SUBAPPLICATION Uebung_060 (* DigitalInput_I1 auf DigitalOutput_Q1 *)
  (* Standard: 61499-2 *)
  (* Version 1.0, 2023-10-23, franz *)
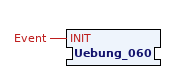
  EVENT_INPUT
    INIT;
  END_EVENT
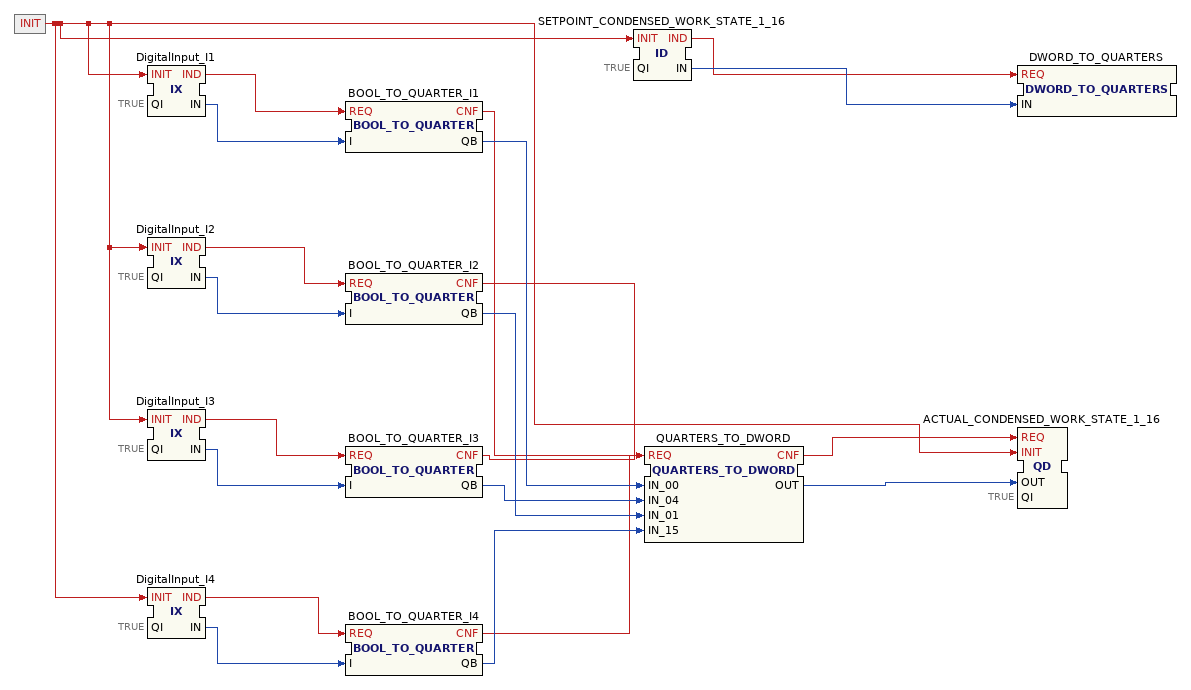
  FBS
    SETPOINT_CONDENSED_WORK_STATE_1_16 : ID(QI := TRUE);
    DWORD_TO_QUARTERS : DWORD_TO_QUARTERS;
    QUARTERS_TO_DWORD : QUARTERS_TO_DWORD;
    ACTUAL_CONDENSED_WORK_STATE_1_16 : QD(QI := TRUE);
    DigitalInput_I1 : IX(QI := TRUE);
    BOOL_TO_QUARTER_I1 : BOOL_TO_QUARTER;
    DigitalInput_I2 : IX(QI := TRUE);
    BOOL_TO_QUARTER_I3 : BOOL_TO_QUARTER;
    DigitalInput_I3 : IX(QI := TRUE);
    DigitalInput_I4 : IX(QI := TRUE);
    BOOL_TO_QUARTER_I2 : BOOL_TO_QUARTER;
    BOOL_TO_QUARTER_I4 : BOOL_TO_QUARTER;
  END_FBS
  EVENT_CONNECTIONS
    INIT TO SETPOINT_CONDENSED_WORK_STATE_1_16.INIT;
    SETPOINT_CONDENSED_WORK_STATE_1_16.IND TO DWORD_TO_QUARTERS.REQ;
    QUARTERS_TO_DWORD.CNF TO ACTUAL_CONDENSED_WORK_STATE_1_16.REQ;
    INIT TO ACTUAL_CONDENSED_WORK_STATE_1_16.INIT;
    INIT TO DigitalInput_I1.INIT;
    DigitalInput_I1.IND TO BOOL_TO_QUARTER_I1.REQ;
    BOOL_TO_QUARTER_I1.CNF TO QUARTERS_TO_DWORD.REQ;
    INIT TO DigitalInput_I2.INIT;
    DigitalInput_I3.IND TO BOOL_TO_QUARTER_I3.REQ;
    BOOL_TO_QUARTER_I3.CNF TO QUARTERS_TO_DWORD.REQ;
    INIT TO DigitalInput_I3.INIT;
    INIT TO DigitalInput_I4.INIT;
    DigitalInput_I2.IND TO BOOL_TO_QUARTER_I2.REQ;
    BOOL_TO_QUARTER_I2.CNF TO QUARTERS_TO_DWORD.REQ;
    DigitalInput_I4.IND TO BOOL_TO_QUARTER_I4.REQ;
    BOOL_TO_QUARTER_I4.CNF TO QUARTERS_TO_DWORD.REQ;
  END_CONNECTIONS
  DATA_CONNECTIONS
    SETPOINT_CONDENSED_WORK_STATE_1_16.IN TO DWORD_TO_QUARTERS.IN;
    QUARTERS_TO_DWORD.OUT TO ACTUAL_CONDENSED_WORK_STATE_1_16.OUT;
    DigitalInput_I1.IN TO BOOL_TO_QUARTER_I1.I;
    BOOL_TO_QUARTER_I1.QB TO QUARTERS_TO_DWORD.IN_00;
    DigitalInput_I3.IN TO BOOL_TO_QUARTER_I3.I;
    BOOL_TO_QUARTER_I3.QB TO QUARTERS_TO_DWORD.IN_04;
    DigitalInput_I2.IN TO BOOL_TO_QUARTER_I2.I;
    BOOL_TO_QUARTER_I2.QB TO QUARTERS_TO_DWORD.IN_01;
    DigitalInput_I4.IN TO BOOL_TO_QUARTER_I4.I;
    BOOL_TO_QUARTER_I4.QB TO QUARTERS_TO_DWORD.IN_15;
  END_CONNECTIONS
END_SUBAPPLICATION
